{attribute 'linkalways'} 
{attribute 'no_explicit_call' := 'This FB is a CLASS and must be accessed using methods or properties'}
{attribute 'enable_dynamic_creation'}
FUNCTION_BLOCK Node_F_VN_FillContainerExp_TcVnVector4_DINT EXTENDS VisionNode
VAR
    ipContainer : _ITcVnContainer;
    aValue : _TcVnVector4_DINT;
    nStartIdx : _ULINT(0);
    nCount : _ULINT(0);
    hrPrev : _HRESULT(S_OK);
    hresult : _HRESULT(S_OK);
END_VAR

METHOD PUBLIC  Clone : I_Node
VAR
    pNode : POINTER TO Node_F_VN_FillContainerExp_TcVnVector4_DINT;
END_VAR
pNode := __NEW(Node_F_VN_FillContainerExp_TcVnVector4_DINT);
Clone := pNode^;
END_METHOD

METHOD FB_init : BOOL
VAR_INPUT
    bInitRetains : BOOL; // if TRUE, the retain variables are initialized (warm start / cold start)
    bInCopyCode : BOOL;  // if TRUE, the instance afterwards gets moved into the copy code (online change)
END_VAR
AddInput('ipContainer', ipContainer);
AddInput('aValue', aValue);
AddInput('nStartIdx', nStartIdx);
AddInput('nCount', nCount);
AddInput('hrPrev', hrPrev);
AddOutput('ipContainer', ipContainer);
AddOutput('hresult',hresult);
END_METHOD

METHOD PROTECTED OnExecute : HRESULT
hresult.Value := F_VN_FillContainerExp_TcVnVector4_DINT(
    ipContainer := ipContainer.Value,
    aValue := aValue.Value,
    nStartIdx := nStartIdx.Value,
    nCount := nCount.Value,
    hrPrev:= hrPrev.Value);
END_METHOD

METHOD PUBLIC PreExecutionCheck
VAR_INPUT
    Check : I_PreExecutionChecks;
END_VAR
Check.IsTrue(ipContainer.IsValid, 'ipContainer must be a valid container');
Check.IsTrue(ipContainer.HasType(TC_GLOBAL_CONST_LIST.ContainerType_Vector_TcVnVector4_DINT), 'ipContainer contains incorrect type');
END_METHOD

END_FUNCTION_BLOCK

(* stored: Version 1.1.0.1, ProductVersion 3.1.4024.13
   POU Node_F_VN_FillContainerExp_TcVnVector4_DINT: Id {dc8ed7f8-b01e-469f-aca4-d1c08aa94b32}, SpecialFunc None
   Folder Constructor: Id {3ef1c59a-5a94-405d-827f-6cb60bdd99cb}
   Method Clone: Id {0a6b3cf7-14cb-46b1-89b1-f3208bfdd26c}
   Method FB_init: Id {dfecb0a5-2ac8-403d-8515-424bf6408312}
   Method OnExecute: Id {fa73438d-6f80-495c-a979-759a37943a4d}
   Method PreExecutionCheck: Id {13732f17-cfe9-4380-9142-b6b0850c1ace} *)
